Universal Robots URScript: 06_var_global_01.script

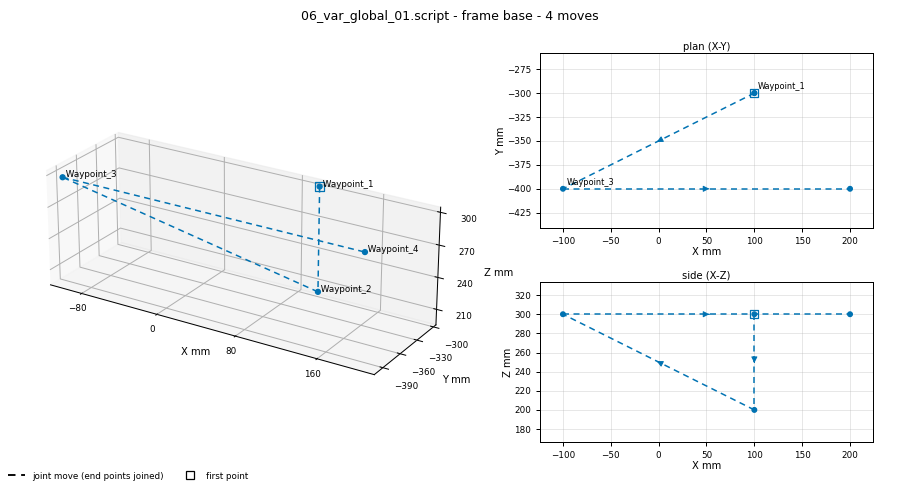
[picture p0: tool path of 06_var_global_01.script in frame base, 4 of 4 moves have a stored position in this frame; points joined in program order, loops and branches not executed]
def P06_var_global_01():
  step_count_77154f07_a93b_4dac_9cdc_12584ce3cc98 = 0.0
  thread Step_Counter_Thread_65f37794_2095_4b5c_a568_ff3977c41b84():
    while (True):
      step_count_77154f07_a93b_4dac_9cdc_12584ce3cc98 = step_count_77154f07_a93b_4dac_9cdc_12584ce3cc98 + 1.0
      sync()
    end
  end
  run Step_Counter_Thread_65f37794_2095_4b5c_a568_ff3977c41b84()
  set_tcp(p[0.0,0.0,0.0,0.0,0.0,0.0])
  set_payload(0.0)
  set_standard_analog_input_domain(0, 1)
  set_standard_analog_input_domain(1, 1)
  set_tool_analog_input_domain(0, 1)
  set_tool_analog_input_domain(1, 1)
  set_analog_outputdomain(0, 0)
  set_analog_outputdomain(1, 0)
  set_input_actions_to_default()
  set_gravity([0.0, 0.0, 9.82])
  set_tool_communication(False, 115200, 0, 1, 1.5, 3.5)
  set_tool_output_mode(0)
  set_tool_digital_output_mode(0, 1)
  set_tool_digital_output_mode(1, 1)
  set_tool_voltage(0)
  set_safety_mode_transition_hardness(1)
  global i_count=1
  global Waypoint_1_p=p[.099999999970, -.300000000017, .299999999988, .001241012500, 3.141592161366, -.000000000274]
  global Waypoint_1_q=[-0.8139121721778135, -1.1456427967711935, -2.388583056583174, -1.1781629571862098, 1.5707965057932782, 0.7576742080001578]
  global Waypoint_2_p=p[.099999999970, -.300000000017, .199999999781, .000000000294, 3.141592162077, .000000000021]
  global Waypoint_2_q=[-0.813912234174393, -1.3594749349082402, -2.5715570584716003, -0.7813566491527046, 1.570796684082526, 0.7568840930129432]
  global Waypoint_3_p=p[-.099999999977, -.399999999988, .299999999988, .000000000294, 3.141592163434, .000000000021]
  global Waypoint_3_q=[-1.486560428667544, -1.4391887816886229, -2.1913789393277145, -1.0818212178987014, 1.570796815459499, 0.08423589851974507]
  global Waypoint_4_p=p[.200000000109, -.399999999988, .299999999988, .000000000294, 3.141592162982, .000000000021]
  global Waypoint_4_q=[-0.8044809343032844, -1.5301612632181731, -2.110032990965097, -1.0721943857764717, 1.5707966800679556, 0.7663153928840454]
  while (True):
    $ 2 "Robot Program"
    $ 3 "MoveJ"
    $ 4 "Waypoint_1" "breakAfter"
    movej(get_inverse_kin(Waypoint_1_p, qnear=Waypoint_1_q), a=1.3962634015954636, v=1.0471975511965976)
    $ 5 "Waypoint_2" "breakAfter"
    movej(get_inverse_kin(Waypoint_2_p, qnear=Waypoint_2_q), a=1.3962634015954636, v=1.0471975511965976)
    $ 6 "Set i_count=i_count+1"
    i_count = i_count + 1
    $ 7 "If i_count≟3"
    if (i_count == 3):
      $ 8 "MoveJ"
      $ 9 "Waypoint_3" "breakAfter"
      movej(get_inverse_kin(Waypoint_3_p, qnear=Waypoint_3_q), a=1.3962634015954636, v=1.0471975511965976)
      $ 10 "Wait: 1.0"
      sleep(1.0)
    end
    $ 11 "If i_count≟5"
    if (i_count == 5):
      $ 12 "MoveJ"
      $ 13 "Waypoint_4" "breakAfter"
      movej(get_inverse_kin(Waypoint_4_p, qnear=Waypoint_4_q), a=1.3962634015954636, v=1.0471975511965976)
      $ 14 "Popup: Jop is done!"
      popup("Jop is done!", "Message", False, False, blocking=True)
      $ 15 "i_count≔0"
      global i_count=0
    end
  end
end
